FUNCTION_BLOCK RobotA22 EXTENDS KukaRobot
VAR_INPUT
	wrapSafety : BOOL;
END_VAR
VAR_OUTPUT //from outputs array
	taskID : TaskA22;
	param1 : INT;
	param2 : INT;
	Xmm : INT;
	Ymm : INT;
	Zmm : INT;
	angle : INT;
	foldPosition0 : INT;
	foldPosition1 : INT;
END_VAR
VAR_OUTPUT //from inputs array
	tool : SectionEnum := SectionEnum.CARDBOARD_CORNERGUARD;
	suspendedMaterial : STRING;
	
	completedTask : TaskA22;
	eoatDistance : INT;
	cardboardAvailability : INT;
	cornerGuardAvailability : INT;
	materialAtHoldingPosition : INT;
	//grp6
	//grp7
	
	wrapSafetyIn : BOOL;
	
END_VAR
VAR //HMI data
	reservationEnum : SectionEnum;
	hmiTask : STRING;
	hmiTool : STRING;
END_VAR

{warning disable C0195}
SUPER^();

outputs[1] := taskID;
outputs[2] := param1;
outputs[3] := param2;
outputs[4] := Xmm;
outputs[5] := Ymm;
outputs[6] := Zmm;
outputs[7] := angle;
outputs[8] := foldPosition0;
outputs[9] := foldPosition1;

refreshParameters();

reservationEnum := reservation;
IF reservationEnum = SectionEnum.NULL_SECTION THEN
	hmiReservation := 'N/A';
ELSE
	hmiReservation := TO_STRING(reservationEnum);
END_IF

hmiTask := TO_STRING(taskID);
hmiTool := TO_STRING(tool);

{attribute 'monitoring' := 'call'}
PROPERTY Busy : BOOL
GET
VAR
	//emptyOutput : ARRAY[1..50] OF INT;
END_VAR
//Busy stays TRUE until outputs are cleared AND completed task has elapsed
//Ready is always inverse of Busy
refreshParameters();

Busy := taskID <> 0 OR completedTask <> 0;
END_GET
END_PROPERTY

METHOD changeEOAT : BOOL
VAR_INPUT
	targetTool : SectionEnum;
END_VAR
//fill in IO here

changeEOAT := TRUE;
END_METHOD

METHOD clearCommand : BOOL
VAR_INPUT
	reserveID : INT;
END_VAR
clearCommand := SUPER^.clearCommand(reserveID := reserveID);

refreshParameters();
END_METHOD

{attribute 'monitoring' := 'call'}
PROPERTY Done : BOOL
GET
refreshParameters();

Done :=
	completedTask = taskID AND
	taskID <> 0 AND
	completedTask <> 0;
END_GET
END_PROPERTY

{attribute 'monitoring' := 'call'}
PROPERTY HoldMaterial : STRING
GET
HoldMaterial := suspendedMaterial;
END_GET
SET
suspendedMaterial := HoldMaterial;
END_SET
END_PROPERTY

{attribute 'monitoring' := 'call'}
PROPERTY Ready : BOOL
GET
refreshParameters();

Ready := taskID = 0 AND completedTask = 0;
END_GET
END_PROPERTY

METHOD PRIVATE refreshParameters : BOOL
VAR_INPUT
END_VAR
{warning disable C0196}
taskID := outputs[1];
param1 := outputs[2];
param2 := outputs[3];
Xmm := outputs[4];
Ymm := outputs[5];
Zmm := outputs[6];
angle := outputs[7];
foldPosition0 := outputs[8];
foldPosition1 := outputs[9];

completedTask := inputs[1];
(*
eoatDistance := inputs[2];
magazineAvailability := inputs[3];
chipboardSkidInPosition := inputs[4];
materialAtHoldingPosition := inputs[5];
//robotEOAT := inputs[6];

strapSafetyIn := inputs[4].15;
*)
END_METHOD

METHOD setGroup : BOOL
VAR_INPUT
	reserveID : INT;
	group : INT;
	value : INT;
END_VAR
SUPER^.setGroup(reserveID := reserveID, group := group, value := value);

refreshParameters();
END_METHOD

METHOD setParameters : BOOL
VAR_INPUT
	reserveID : INT;
	
	newTaskID : INT;
	newParam1 : INT;
	newParam2 : INT;
	newXmm : INT;
	newYmm : INT;
	newZmm : INT;
	newAngle : INT;
	newStagingOccupancy : INT;
	newInsertionSuctionStatus : INT;
	newMagazineStatus : INT; //unused
	newInspectionValue : INT;
END_VAR
setGroup(reserveID := reserveID, group := 1, value := newTaskID);
setGroup(reserveID := reserveID, group := 2, value := newParam1);
setGroup(reserveID := reserveID, group := 3, value := newParam2);
setGroup(reserveID := reserveID, group := 4, value := newXmm);
setGroup(reserveID := reserveID, group := 5, value := newYmm);
setGroup(reserveID := reserveID, group := 6, value := newZmm);
setGroup(reserveID := reserveID, group := 7, value := newAngle);

newStagingOccupancy.15 := wrapSafety;
setGroup(reserveID := reserveID, group := 8, value := newStagingOccupancy);

setGroup(reserveID := reserveID, group := 9, value := newInsertionSuctionStatus);
setGroup(reserveID := reserveID, group := 10, value := newMagazineStatus);
setGroup(reserveID := reserveID, group := 11, value := newInspectionValue);

refreshParameters();
END_METHOD

END_FUNCTION_BLOCK

(* stored: Version 1.1.0.1, ProductVersion 3.1.4024.11
   POU RobotA22: Id {870b17d8-8fed-45ea-b532-f3f727b3e8ec}, SpecialFunc None
   Folder Parameters: Id {f09709b6-ac88-41fd-a494-6ff3c05edd5a}
   Folder Properties: Id {dc127a71-2b3d-47e3-acd0-c3047f90d92c}
   Property Busy: Id {51e7c5e7-986b-486d-a66a-1d713a8b811d}
   Get Get: Id {20dcedf2-865e-4b4a-b529-a2cc2e87f1a8}
   Method changeEOAT: Id {5c591e9f-42b5-4ae1-b808-b0e182093d21}
   Method clearCommand: Id {29dd27f6-3ae8-479e-9b8d-f4f10f6725b3}
   Property Done: Id {8cc7b7f2-6ad0-499f-81d6-95864fbc7677}
   Get Get: Id {b47f3d65-5556-4732-887f-a8687173a85f}
   Property HoldMaterial: Id {7e43bb07-0140-4b4a-903a-aa723ec40da6}
   Get Get: Id {a9326765-7208-4d2c-93bc-2fbdd9a9791d}
   Set Set: Id {57c07f37-cab4-4e43-884f-dbb4a5b2fc77}
   Property Ready: Id {12815c93-fa28-4f21-b13f-9c71481b0999}
   Get Get: Id {342973ce-41eb-4aff-85e7-0c033c6d77c0}
   Method refreshParameters: Id {278c3745-7dcb-41fb-a68e-c0fbaeb86786}
   Method setGroup: Id {0c432c8e-49f0-4570-9f83-a738dd9919d8}
   Method setParameters: Id {9c320439-85d7-4395-a3ec-b5d8cea0aeff} *)
